// TIA Portal V19 export
VAR_GLOBAL   // PLC tag table "U3Em0_input"
END_VAR
